// TIA Portal V17 export
// export: Created 2025-03-18T12:31:00.4756631Z, ExportSetting WithDefaults, DisplayName Totally Integrated Automation Portal, DisplayVersion V17 Update 8, DisplayName TIA Portal Openness, DisplayVersion V17 Update 8, DisplayName TIA Portal Version Control Interface, DisplayVersion V17, DisplayName SINAMICS Startdrive Advanced, DisplayVersion V17 SP2, DisplayName SINAMICS Startdrive G110M, G120, G120C, G120D, G120P, G115D, DisplayVersion V17 SP2, DisplayName SINAMICS Startdrive G130, G150, S120, S150, SINAMICS MV, S210, DisplayVersion V17 SP2, DisplayName STEP 7 Professional, DisplayVersion V17 Update 8, DisplayName SINUMERIK ONE STEP 7 Toolbox, DisplayVersion V17 Update 12, DisplayName SINUMERIK 840D sl STEP 7 Toolbox, DisplayVersion V17 Update 12, DisplayName STEP 7 Safety, DisplayVersion V17 Update 6, DisplayName WinCC Advanced, DisplayVersion V17 Update 8
FUNCTION "FC7003_UNIT_01_STATION_04_SAFETY_DOOR" : Void   // FC7003, LAD
{ S7_Optimized_Access := 'FALSE' }
AUTHOR : ETXETAR
VERSION : 1.0
// stored: AutoNumber false, IsIECCheckEnabled false, SetENOAutomatically false, UDAEnableTagReadback false
   VAR_INPUT
      OPTIONS_0 : Byte;   // OPTIONS 0
      CLOSED : Bool;   // CLOSED INPUT
      LOCKED : Bool;   // LOCKED INPUT
   END_VAR
   VAR_OUTPUT
      UNLOCK : Bool;   // UNLOCK OUTPUT
      RED_LIGTH : Bool;   // RED LIGTH OUTPUT
      GREEN_LIGTH : Bool;   // GREEN LIGTH OUTPUT
   END_VAR
   VAR_TEMP
      INPUTS_MASK : Byte;   // INPUTS MASK
      O_BYTE_0 : Struct   // OPTIONS BYTE 0
         IMMEDIATE_STOP : Bool;   // IMMEDIATE STOP REACTION OPTION
         SEOC_WARNING : Bool;   // SEOC WARNING REACTION OPTION
         CLOSED_SENSOR_I : Bool;   // CLOSED SENSOR INPUT OPTION
         CIRCUIT_E2 : Bool;   // CIRCUIT E2 OPTION
         PNEUMATIC_DRIVE : Bool;   // PNEUMATIC DRIVE OPTION
         CHIP_CONVEYOR : Bool;   // CHIP CONVEYOR OPTION
         SPARE_6 : Bool;   // SPARE OPTION
         SPARE_7 : Bool;   // SPARE OPTION
      END_STRUCT;
   END_VAR
   VAR CONSTANT
      FC_NUMBER : DInt := 7003;
   END_VAR
   VAR_TEMP   // added for the SCL form of the ladder/FBD networks
      _w1 : Bool;
      _w2 : Bool;
   END_VAR
BEGIN

REGION Network 1: OPTIONS
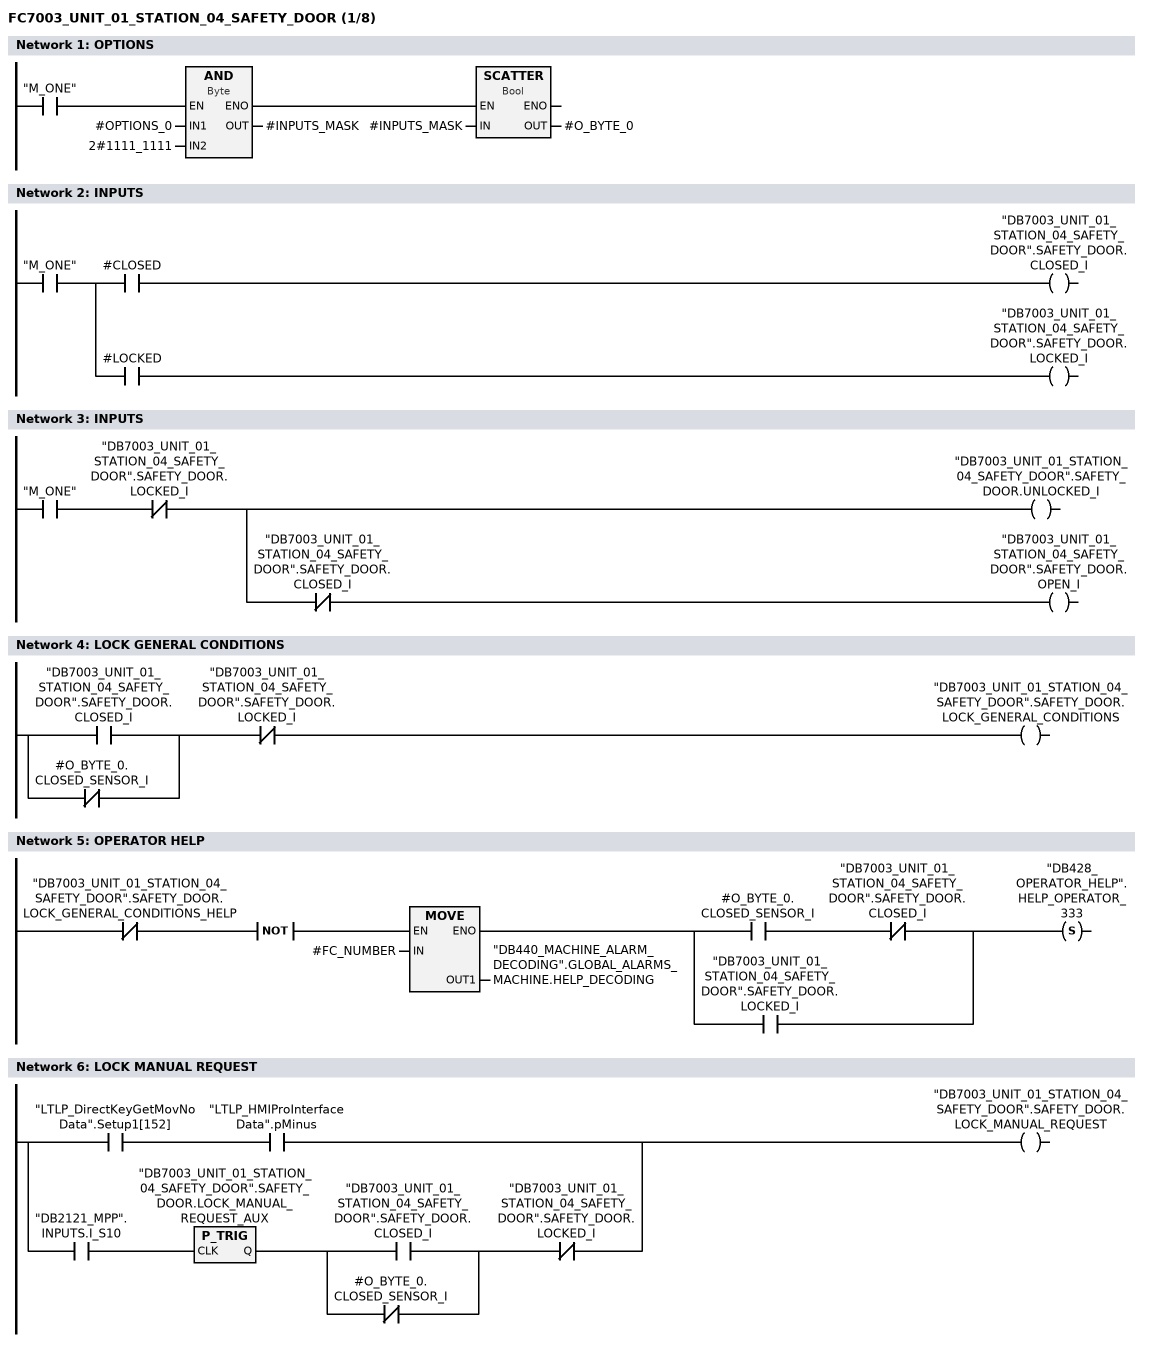
   RUNG wire#powerrail
      Contact( "M_ONE" )
      { S7_Templates := "SrcType := Byte"; S7_GenerateENO := "TRUE" } And(in1 := #OPTIONS_0, in2 := 2#1111_1111, out => #INPUTS_MASK)
      { S7_Templates := "[dest_type := Bool, src_type := Byte]" } SCATTER(IN := #INPUTS_MASK, OUT => #O_BYTE_0)
   END_RUNG
   // the same network as SCL:
   IF "M_ONE" THEN
       #INPUTS_MASK := #OPTIONS_0 AND 2#1111_1111;
       SCATTER(IN := #INPUTS_MASK, OUT => #O_BYTE_0);
   END_IF;
END_REGION

REGION Network 2: INPUTS
   RUNG wire#powerrail
      Contact( "M_ONE" )
      wire#w1
      Contact( #CLOSED )
      Coil( "DB7003_UNIT_01_STATION_04_SAFETY_DOOR".SAFETY_DOOR.CLOSED_I )
   END_RUNG
   RUNG wire#w1
      Contact( #LOCKED )
      Coil( "DB7003_UNIT_01_STATION_04_SAFETY_DOOR".SAFETY_DOOR.LOCKED_I )
   END_RUNG
   // the same network as SCL:
   "DB7003_UNIT_01_STATION_04_SAFETY_DOOR".SAFETY_DOOR.CLOSED_I := "M_ONE" AND #CLOSED;
   "DB7003_UNIT_01_STATION_04_SAFETY_DOOR".SAFETY_DOOR.LOCKED_I := "M_ONE" AND #LOCKED;
END_REGION

REGION Network 3: INPUTS
   RUNG wire#powerrail
      Contact( "M_ONE" )
      I_Contact( "DB7003_UNIT_01_STATION_04_SAFETY_DOOR".SAFETY_DOOR.LOCKED_I )
      wire#w1
      Coil( "DB7003_UNIT_01_STATION_04_SAFETY_DOOR".SAFETY_DOOR.UNLOCKED_I )
   END_RUNG
   RUNG wire#w1
      I_Contact( "DB7003_UNIT_01_STATION_04_SAFETY_DOOR".SAFETY_DOOR.CLOSED_I )
      Coil( "DB7003_UNIT_01_STATION_04_SAFETY_DOOR".SAFETY_DOOR.OPEN_I )
   END_RUNG
   // the same network as SCL:
   "DB7003_UNIT_01_STATION_04_SAFETY_DOOR".SAFETY_DOOR.UNLOCKED_I := "M_ONE" AND NOT "DB7003_UNIT_01_STATION_04_SAFETY_DOOR".SAFETY_DOOR.LOCKED_I;
   "DB7003_UNIT_01_STATION_04_SAFETY_DOOR".SAFETY_DOOR.OPEN_I := "DB7003_UNIT_01_STATION_04_SAFETY_DOOR".SAFETY_DOOR.UNLOCKED_I AND NOT "DB7003_UNIT_01_STATION_04_SAFETY_DOOR".SAFETY_DOOR.CLOSED_I;
END_REGION

REGION Network 4: LOCK GENERAL CONDITIONS
   RUNG wire#powerrail
      Contact( "DB7003_UNIT_01_STATION_04_SAFETY_DOOR".SAFETY_DOOR.CLOSED_I )
      wire#w1
      I_Contact( "DB7003_UNIT_01_STATION_04_SAFETY_DOOR".SAFETY_DOOR.LOCKED_I )
      Coil( "DB7003_UNIT_01_STATION_04_SAFETY_DOOR".SAFETY_DOOR.LOCK_GENERAL_CONDITIONS )
   END_RUNG
   RUNG wire#powerrail
      I_Contact( #O_BYTE_0.CLOSED_SENSOR_I )
   END_RUNG wire#w1
   // the same network as SCL:
   "DB7003_UNIT_01_STATION_04_SAFETY_DOOR".SAFETY_DOOR.LOCK_GENERAL_CONDITIONS := ("DB7003_UNIT_01_STATION_04_SAFETY_DOOR".SAFETY_DOOR.CLOSED_I OR NOT #O_BYTE_0.CLOSED_SENSOR_I) AND NOT "DB7003_UNIT_01_STATION_04_SAFETY_DOOR".SAFETY_DOOR.LOCKED_I;
END_REGION

REGION Network 5: OPERATOR HELP
   RUNG wire#powerrail
      I_Contact( "DB7003_UNIT_01_STATION_04_SAFETY_DOOR".SAFETY_DOOR.LOCK_GENERAL_CONDITIONS_HELP )
      Not()
      { S7_GenerateENO := "TRUE" } Move(in := #FC_NUMBER, out1 => "DB440_MACHINE_ALARM_DECODING".GLOBAL_ALARMS_MACHINE.HELP_DECODING)
      wire#w1
      Contact( #O_BYTE_0.CLOSED_SENSOR_I )
      I_Contact( "DB7003_UNIT_01_STATION_04_SAFETY_DOOR".SAFETY_DOOR.CLOSED_I )
      wire#w2
      S_Coil( "DB428_OPERATOR_HELP".HELP_OPERATOR_333 )
   END_RUNG
   RUNG wire#w1
      Contact( "DB7003_UNIT_01_STATION_04_SAFETY_DOOR".SAFETY_DOOR.LOCKED_I )
   END_RUNG wire#w2
   // the same network as SCL:
   // ENO of a box is taken as its EN; it also drops when the box reports an error
   #_w1 := NOT (NOT "DB7003_UNIT_01_STATION_04_SAFETY_DOOR".SAFETY_DOOR.LOCK_GENERAL_CONDITIONS_HELP);
   IF #_w1 THEN "DB440_MACHINE_ALARM_DECODING".GLOBAL_ALARMS_MACHINE.HELP_DECODING := #FC_NUMBER; END_IF;
   IF #_w1 AND ((#O_BYTE_0.CLOSED_SENSOR_I AND NOT "DB7003_UNIT_01_STATION_04_SAFETY_DOOR".SAFETY_DOOR.CLOSED_I) OR "DB7003_UNIT_01_STATION_04_SAFETY_DOOR".SAFETY_DOOR.LOCKED_I) THEN
       "DB428_OPERATOR_HELP".HELP_OPERATOR_333 := TRUE;
   END_IF;
END_REGION

REGION Network 6: LOCK MANUAL REQUEST
   RUNG wire#powerrail
      Contact( "LTLP_DirectKeyGetMovNoData".Setup1[152] )
      Contact( "LTLP_HMIProInterfaceData".pMinus )
      wire#w1
      Coil( "DB7003_UNIT_01_STATION_04_SAFETY_DOOR".SAFETY_DOOR.LOCK_MANUAL_REQUEST )
   END_RUNG
   RUNG wire#powerrail
      Contact( "DB2121_MPP".INPUTS.I_S10 )
      P_Trig( "DB7003_UNIT_01_STATION_04_SAFETY_DOOR".SAFETY_DOOR.LOCK_MANUAL_REQUEST_AUX )
      wire#w2
      Contact( "DB7003_UNIT_01_STATION_04_SAFETY_DOOR".SAFETY_DOOR.CLOSED_I )
      wire#w3
      I_Contact( "DB7003_UNIT_01_STATION_04_SAFETY_DOOR".SAFETY_DOOR.LOCKED_I )
   END_RUNG wire#w1
   RUNG wire#w2
      I_Contact( #O_BYTE_0.CLOSED_SENSOR_I )
   END_RUNG wire#w3
   // the same network as SCL:
   #_w1 := "DB2121_MPP".INPUTS.I_S10 AND NOT "DB7003_UNIT_01_STATION_04_SAFETY_DOOR".SAFETY_DOOR.LOCK_MANUAL_REQUEST_AUX;   // rising edge
   "DB7003_UNIT_01_STATION_04_SAFETY_DOOR".SAFETY_DOOR.LOCK_MANUAL_REQUEST_AUX := "DB2121_MPP".INPUTS.I_S10;
   "DB7003_UNIT_01_STATION_04_SAFETY_DOOR".SAFETY_DOOR.LOCK_MANUAL_REQUEST := ("LTLP_DirectKeyGetMovNoData".Setup1[152] AND "LTLP_HMIProInterfaceData".pMinus) OR (#_w1 AND ("DB7003_UNIT_01_STATION_04_SAFETY_DOOR".SAFETY_DOOR.CLOSED_I OR NOT #O_BYTE_0.CLOSED_SENSOR_I) AND NOT "DB7003_UNIT_01_STATION_04_SAFETY_DOOR".SAFETY_DOOR.LOCKED_I);
END_REGION

REGION Network 7: LOCK AUTO REQUEST
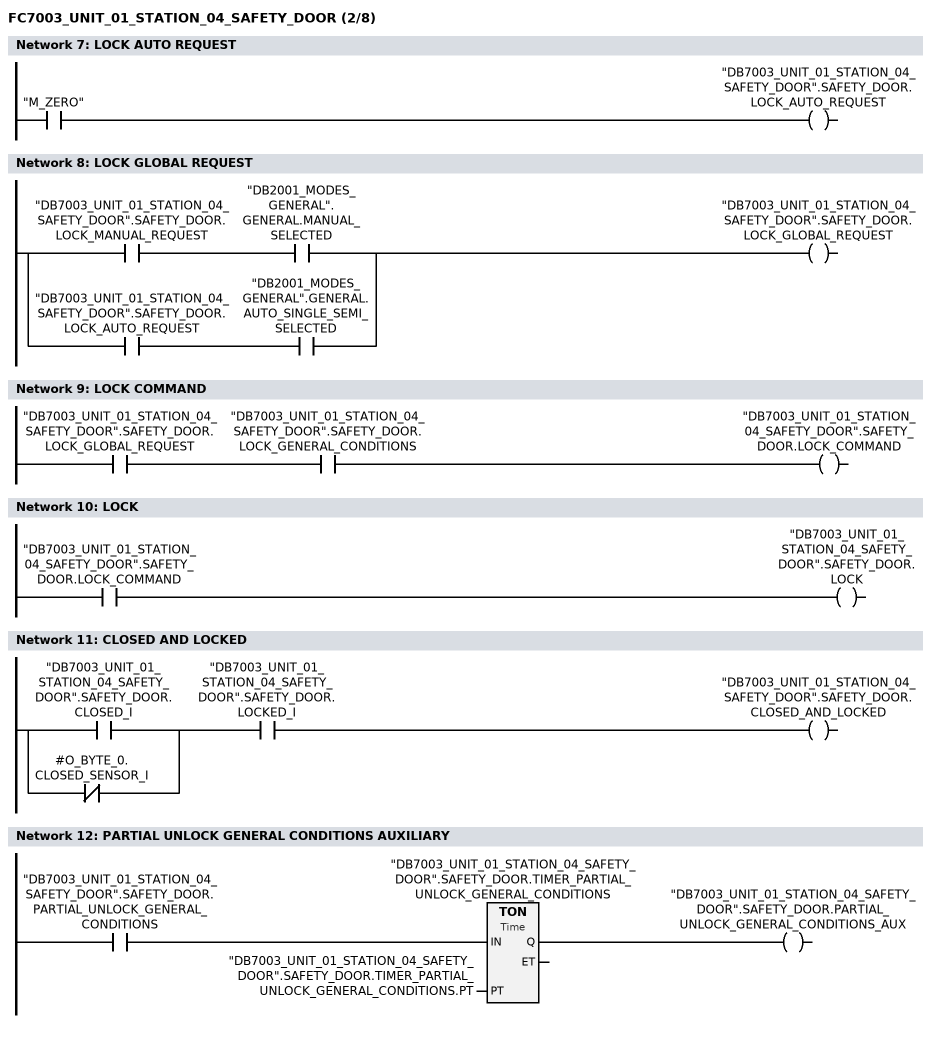
   RUNG wire#powerrail
      Contact( "M_ZERO" )
      Coil( "DB7003_UNIT_01_STATION_04_SAFETY_DOOR".SAFETY_DOOR.LOCK_AUTO_REQUEST )
   END_RUNG
   // the same network as SCL:
   "DB7003_UNIT_01_STATION_04_SAFETY_DOOR".SAFETY_DOOR.LOCK_AUTO_REQUEST := "M_ZERO";
END_REGION

REGION Network 8: LOCK GLOBAL REQUEST
   RUNG wire#powerrail
      Contact( "DB7003_UNIT_01_STATION_04_SAFETY_DOOR".SAFETY_DOOR.LOCK_MANUAL_REQUEST )
      Contact( "DB2001_MODES_GENERAL".GENERAL.MANUAL_SELECTED )
      wire#w1
      Coil( "DB7003_UNIT_01_STATION_04_SAFETY_DOOR".SAFETY_DOOR.LOCK_GLOBAL_REQUEST )
   END_RUNG
   RUNG wire#powerrail
      Contact( "DB7003_UNIT_01_STATION_04_SAFETY_DOOR".SAFETY_DOOR.LOCK_AUTO_REQUEST )
      Contact( "DB2001_MODES_GENERAL".GENERAL.AUTO_SINGLE_SEMI_SELECTED )
   END_RUNG wire#w1
   // the same network as SCL:
   "DB7003_UNIT_01_STATION_04_SAFETY_DOOR".SAFETY_DOOR.LOCK_GLOBAL_REQUEST := ("DB7003_UNIT_01_STATION_04_SAFETY_DOOR".SAFETY_DOOR.LOCK_MANUAL_REQUEST AND "DB2001_MODES_GENERAL".GENERAL.MANUAL_SELECTED) OR ("DB7003_UNIT_01_STATION_04_SAFETY_DOOR".SAFETY_DOOR.LOCK_AUTO_REQUEST AND "DB2001_MODES_GENERAL".GENERAL.AUTO_SINGLE_SEMI_SELECTED);
END_REGION

REGION Network 9: LOCK COMMAND
   RUNG wire#powerrail
      Contact( "DB7003_UNIT_01_STATION_04_SAFETY_DOOR".SAFETY_DOOR.LOCK_GLOBAL_REQUEST )
      Contact( "DB7003_UNIT_01_STATION_04_SAFETY_DOOR".SAFETY_DOOR.LOCK_GENERAL_CONDITIONS )
      Coil( "DB7003_UNIT_01_STATION_04_SAFETY_DOOR".SAFETY_DOOR.LOCK_COMMAND )
   END_RUNG
   // the same network as SCL:
   "DB7003_UNIT_01_STATION_04_SAFETY_DOOR".SAFETY_DOOR.LOCK_COMMAND := "DB7003_UNIT_01_STATION_04_SAFETY_DOOR".SAFETY_DOOR.LOCK_GLOBAL_REQUEST AND "DB7003_UNIT_01_STATION_04_SAFETY_DOOR".SAFETY_DOOR.LOCK_GENERAL_CONDITIONS;
END_REGION

REGION Network 10: LOCK
   RUNG wire#powerrail
      Contact( "DB7003_UNIT_01_STATION_04_SAFETY_DOOR".SAFETY_DOOR.LOCK_COMMAND )
      Coil( "DB7003_UNIT_01_STATION_04_SAFETY_DOOR".SAFETY_DOOR.LOCK )
   END_RUNG
   // the same network as SCL:
   "DB7003_UNIT_01_STATION_04_SAFETY_DOOR".SAFETY_DOOR.LOCK := "DB7003_UNIT_01_STATION_04_SAFETY_DOOR".SAFETY_DOOR.LOCK_COMMAND;
END_REGION

REGION Network 11: CLOSED AND LOCKED
   RUNG wire#powerrail
      Contact( "DB7003_UNIT_01_STATION_04_SAFETY_DOOR".SAFETY_DOOR.CLOSED_I )
      wire#w1
      Contact( "DB7003_UNIT_01_STATION_04_SAFETY_DOOR".SAFETY_DOOR.LOCKED_I )
      Coil( "DB7003_UNIT_01_STATION_04_SAFETY_DOOR".SAFETY_DOOR.CLOSED_AND_LOCKED )
   END_RUNG
   RUNG wire#powerrail
      I_Contact( #O_BYTE_0.CLOSED_SENSOR_I )
   END_RUNG wire#w1
   // the same network as SCL:
   "DB7003_UNIT_01_STATION_04_SAFETY_DOOR".SAFETY_DOOR.CLOSED_AND_LOCKED := ("DB7003_UNIT_01_STATION_04_SAFETY_DOOR".SAFETY_DOOR.CLOSED_I OR NOT #O_BYTE_0.CLOSED_SENSOR_I) AND "DB7003_UNIT_01_STATION_04_SAFETY_DOOR".SAFETY_DOOR.LOCKED_I;
END_REGION

REGION Network 12: PARTIAL UNLOCK GENERAL CONDITIONS AUXILIARY
   RUNG wire#powerrail
      Contact( "DB7003_UNIT_01_STATION_04_SAFETY_DOOR".SAFETY_DOOR.PARTIAL_UNLOCK_GENERAL_CONDITIONS )
      { S7_Templates := "time_type := Time" } "DB7003_UNIT_01_STATION_04_SAFETY_DOOR".SAFETY_DOOR.TIMER_PARTIAL_UNLOCK_GENERAL_CONDITIONS.TON(pt := "DB7003_UNIT_01_STATION_04_SAFETY_DOOR".SAFETY_DOOR.TIMER_PARTIAL_UNLOCK_GENERAL_CONDITIONS.PT, et =>)
      Coil( "DB7003_UNIT_01_STATION_04_SAFETY_DOOR".SAFETY_DOOR.PARTIAL_UNLOCK_GENERAL_CONDITIONS_AUX )
   END_RUNG
   // the same network as SCL:
   "DB7003_UNIT_01_STATION_04_SAFETY_DOOR".SAFETY_DOOR.TIMER_PARTIAL_UNLOCK_GENERAL_CONDITIONS.TON(IN := "DB7003_UNIT_01_STATION_04_SAFETY_DOOR".SAFETY_DOOR.PARTIAL_UNLOCK_GENERAL_CONDITIONS,
                           PT := "DB7003_UNIT_01_STATION_04_SAFETY_DOOR".SAFETY_DOOR.TIMER_PARTIAL_UNLOCK_GENERAL_CONDITIONS.PT);
   "DB7003_UNIT_01_STATION_04_SAFETY_DOOR".SAFETY_DOOR.PARTIAL_UNLOCK_GENERAL_CONDITIONS_AUX := "DB7003_UNIT_01_STATION_04_SAFETY_DOOR".SAFETY_DOOR.TIMER_PARTIAL_UNLOCK_GENERAL_CONDITIONS.Q;
END_REGION

REGION Network 13: UNLOCK GENERAL CONDITIONS
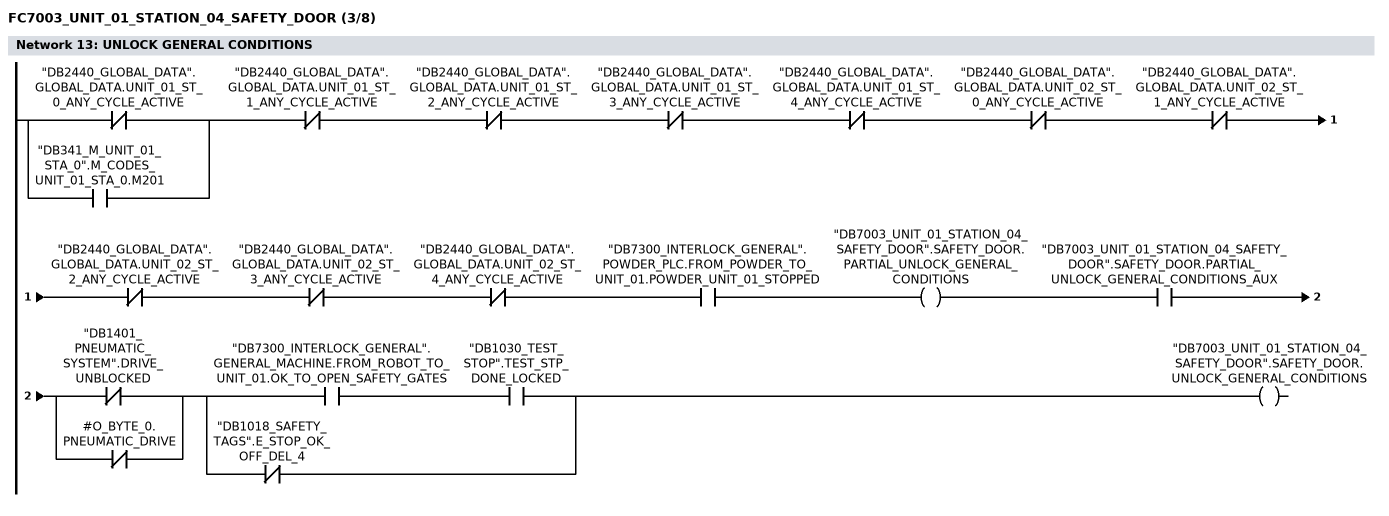
   RUNG wire#powerrail
      I_Contact( "DB2440_GLOBAL_DATA".GLOBAL_DATA.UNIT_01_ST_0_ANY_CYCLE_ACTIVE )
      wire#w1
      I_Contact( "DB2440_GLOBAL_DATA".GLOBAL_DATA.UNIT_01_ST_1_ANY_CYCLE_ACTIVE )
      I_Contact( "DB2440_GLOBAL_DATA".GLOBAL_DATA.UNIT_01_ST_2_ANY_CYCLE_ACTIVE )
      I_Contact( "DB2440_GLOBAL_DATA".GLOBAL_DATA.UNIT_01_ST_3_ANY_CYCLE_ACTIVE )
      I_Contact( "DB2440_GLOBAL_DATA".GLOBAL_DATA.UNIT_01_ST_4_ANY_CYCLE_ACTIVE )
      I_Contact( "DB2440_GLOBAL_DATA".GLOBAL_DATA.UNIT_02_ST_0_ANY_CYCLE_ACTIVE )
      I_Contact( "DB2440_GLOBAL_DATA".GLOBAL_DATA.UNIT_02_ST_1_ANY_CYCLE_ACTIVE )
      I_Contact( "DB2440_GLOBAL_DATA".GLOBAL_DATA.UNIT_02_ST_2_ANY_CYCLE_ACTIVE )
      I_Contact( "DB2440_GLOBAL_DATA".GLOBAL_DATA.UNIT_02_ST_3_ANY_CYCLE_ACTIVE )
      I_Contact( "DB2440_GLOBAL_DATA".GLOBAL_DATA.UNIT_02_ST_4_ANY_CYCLE_ACTIVE )
      Contact( "DB7300_INTERLOCK_GENERAL".POWDER_PLC.FROM_POWDER_TO_UNIT_01.POWDER_UNIT_01_STOPPED )
      Coil( "DB7003_UNIT_01_STATION_04_SAFETY_DOOR".SAFETY_DOOR.PARTIAL_UNLOCK_GENERAL_CONDITIONS )
      Contact( "DB7003_UNIT_01_STATION_04_SAFETY_DOOR".SAFETY_DOOR.PARTIAL_UNLOCK_GENERAL_CONDITIONS_AUX )
      wire#w2
      I_Contact( "DB1401_PNEUMATIC_SYSTEM".DRIVE_UNBLOCKED )
      wire#w3
      Contact( "DB7300_INTERLOCK_GENERAL".GENERAL_MACHINE.FROM_ROBOT_TO_UNIT_01.OK_TO_OPEN_SAFETY_GATES )
      Contact( "DB1030_TEST_STOP".TEST_STP_DONE_LOCKED )
      wire#w4
      Coil( "DB7003_UNIT_01_STATION_04_SAFETY_DOOR".SAFETY_DOOR.UNLOCK_GENERAL_CONDITIONS )
   END_RUNG
   RUNG wire#powerrail
      Contact( "DB341_M_UNIT_01_STA_0".M_CODES_UNIT_01_STA_0.M201 )
   END_RUNG wire#w1
   RUNG wire#w2
      I_Contact( #O_BYTE_0.PNEUMATIC_DRIVE )
   END_RUNG wire#w3
   RUNG wire#w3
      I_Contact( "DB1018_SAFETY_TAGS".E_STOP_OK_OFF_DEL_4 )
   END_RUNG wire#w4
   // the same network as SCL:
   "DB7003_UNIT_01_STATION_04_SAFETY_DOOR".SAFETY_DOOR.PARTIAL_UNLOCK_GENERAL_CONDITIONS := (NOT "DB2440_GLOBAL_DATA".GLOBAL_DATA.UNIT_01_ST_0_ANY_CYCLE_ACTIVE OR "DB341_M_UNIT_01_STA_0".M_CODES_UNIT_01_STA_0.M201) AND NOT "DB2440_GLOBAL_DATA".GLOBAL_DATA.UNIT_01_ST_1_ANY_CYCLE_ACTIVE AND NOT "DB2440_GLOBAL_DATA".GLOBAL_DATA.UNIT_01_ST_2_ANY_CYCLE_ACTIVE AND NOT "DB2440_GLOBAL_DATA".GLOBAL_DATA.UNIT_01_ST_3_ANY_CYCLE_ACTIVE AND NOT "DB2440_GLOBAL_DATA".GLOBAL_DATA.UNIT_01_ST_4_ANY_CYCLE_ACTIVE AND NOT "DB2440_GLOBAL_DATA".GLOBAL_DATA.UNIT_02_ST_0_ANY_CYCLE_ACTIVE AND NOT "DB2440_GLOBAL_DATA".GLOBAL_DATA.UNIT_02_ST_1_ANY_CYCLE_ACTIVE AND NOT "DB2440_GLOBAL_DATA".GLOBAL_DATA.UNIT_02_ST_2_ANY_CYCLE_ACTIVE AND NOT "DB2440_GLOBAL_DATA".GLOBAL_DATA.UNIT_02_ST_3_ANY_CYCLE_ACTIVE AND NOT "DB2440_GLOBAL_DATA".GLOBAL_DATA.UNIT_02_ST_4_ANY_CYCLE_ACTIVE AND "DB7300_INTERLOCK_GENERAL".POWDER_PLC.FROM_POWDER_TO_UNIT_01.POWDER_UNIT_01_STOPPED;
   "DB7003_UNIT_01_STATION_04_SAFETY_DOOR".SAFETY_DOOR.UNLOCK_GENERAL_CONDITIONS := "DB7003_UNIT_01_STATION_04_SAFETY_DOOR".SAFETY_DOOR.PARTIAL_UNLOCK_GENERAL_CONDITIONS AND "DB7003_UNIT_01_STATION_04_SAFETY_DOOR".SAFETY_DOOR.PARTIAL_UNLOCK_GENERAL_CONDITIONS_AUX AND (NOT "DB1401_PNEUMATIC_SYSTEM".DRIVE_UNBLOCKED OR NOT #O_BYTE_0.PNEUMATIC_DRIVE) AND (("DB7300_INTERLOCK_GENERAL".GENERAL_MACHINE.FROM_ROBOT_TO_UNIT_01.OK_TO_OPEN_SAFETY_GATES AND "DB1030_TEST_STOP".TEST_STP_DONE_LOCKED) OR NOT "DB1018_SAFETY_TAGS".E_STOP_OK_OFF_DEL_4);
END_REGION

REGION Network 14: OPERATOR HELP
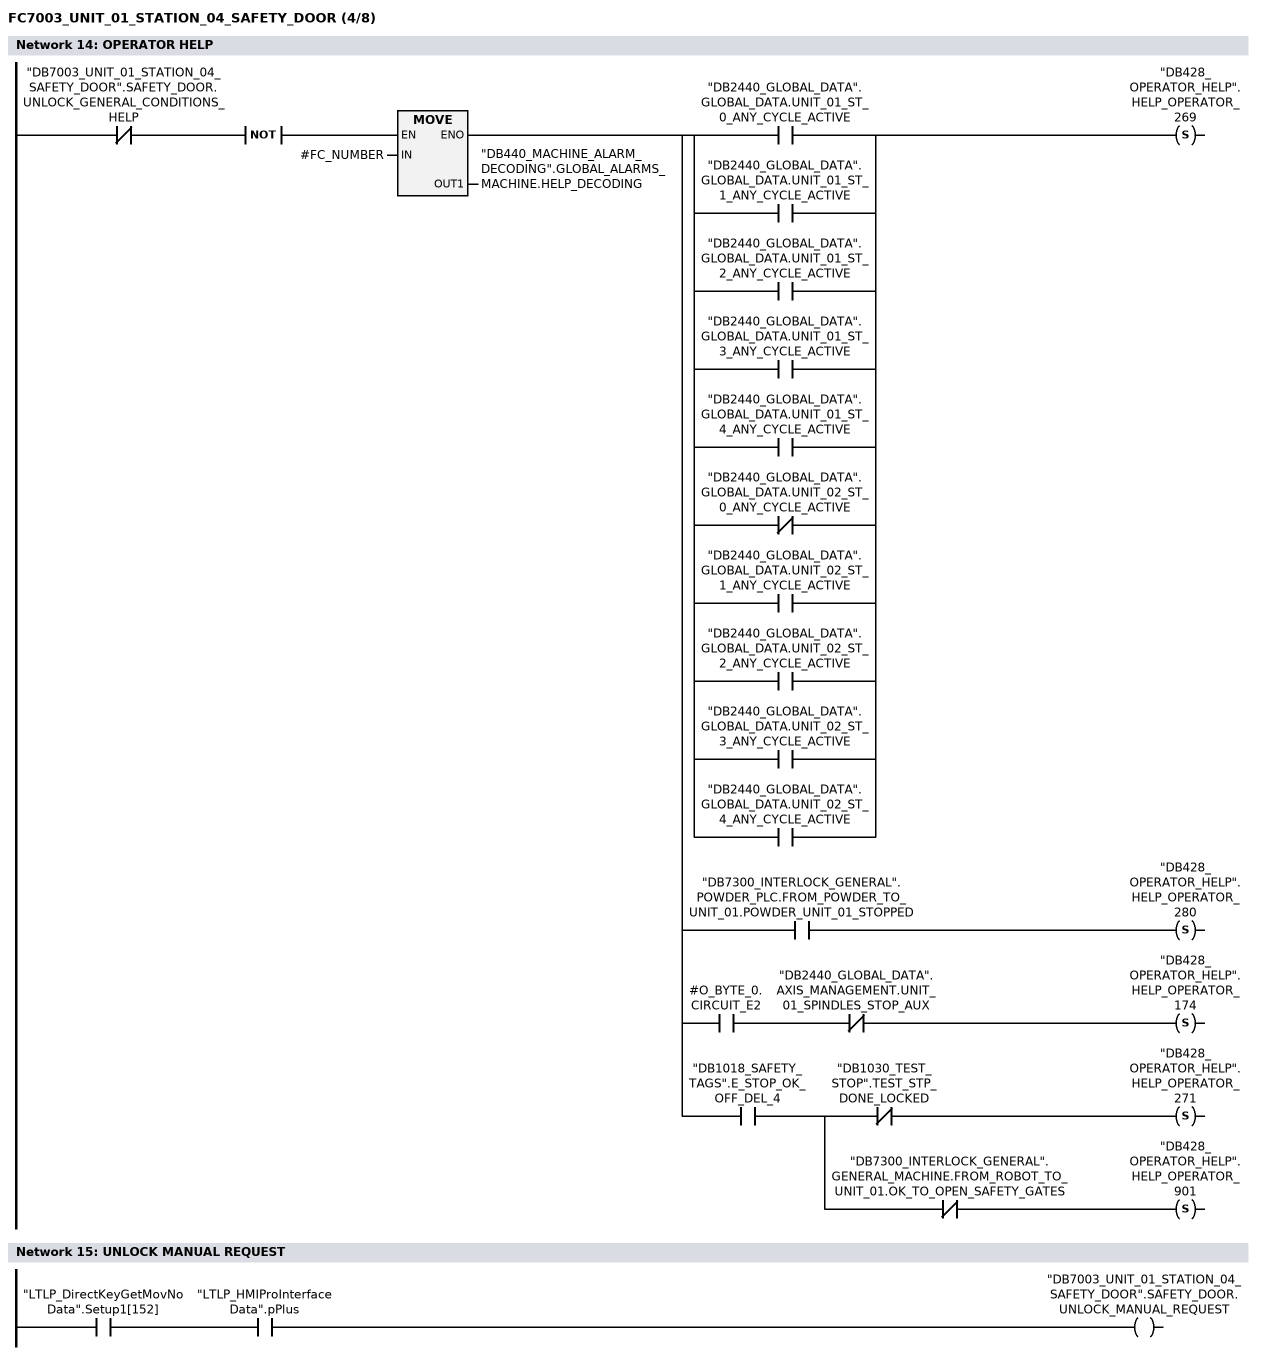
   RUNG wire#powerrail
      I_Contact( "DB7003_UNIT_01_STATION_04_SAFETY_DOOR".SAFETY_DOOR.UNLOCK_GENERAL_CONDITIONS_HELP )
      Not()
      { S7_GenerateENO := "TRUE" } Move(in := #FC_NUMBER, out1 => "DB440_MACHINE_ALARM_DECODING".GLOBAL_ALARMS_MACHINE.HELP_DECODING)
      wire#w1
      Contact( "DB2440_GLOBAL_DATA".GLOBAL_DATA.UNIT_01_ST_0_ANY_CYCLE_ACTIVE )
      wire#w2
      S_Coil( "DB428_OPERATOR_HELP".HELP_OPERATOR_269 )
   END_RUNG
   RUNG wire#w1
      Contact( "DB2440_GLOBAL_DATA".GLOBAL_DATA.UNIT_01_ST_1_ANY_CYCLE_ACTIVE )
   END_RUNG wire#w2
   RUNG wire#w1
      Contact( "DB2440_GLOBAL_DATA".GLOBAL_DATA.UNIT_01_ST_2_ANY_CYCLE_ACTIVE )
   END_RUNG wire#w2
   RUNG wire#w1
      Contact( "DB2440_GLOBAL_DATA".GLOBAL_DATA.UNIT_01_ST_3_ANY_CYCLE_ACTIVE )
   END_RUNG wire#w2
   RUNG wire#w1
      Contact( "DB2440_GLOBAL_DATA".GLOBAL_DATA.UNIT_01_ST_4_ANY_CYCLE_ACTIVE )
   END_RUNG wire#w2
   RUNG wire#w1
      I_Contact( "DB2440_GLOBAL_DATA".GLOBAL_DATA.UNIT_02_ST_0_ANY_CYCLE_ACTIVE )
   END_RUNG wire#w2
   RUNG wire#w1
      Contact( "DB2440_GLOBAL_DATA".GLOBAL_DATA.UNIT_02_ST_1_ANY_CYCLE_ACTIVE )
   END_RUNG wire#w2
   RUNG wire#w1
      Contact( "DB2440_GLOBAL_DATA".GLOBAL_DATA.UNIT_02_ST_2_ANY_CYCLE_ACTIVE )
   END_RUNG wire#w2
   RUNG wire#w1
      Contact( "DB2440_GLOBAL_DATA".GLOBAL_DATA.UNIT_02_ST_3_ANY_CYCLE_ACTIVE )
   END_RUNG wire#w2
   RUNG wire#w1
      Contact( "DB2440_GLOBAL_DATA".GLOBAL_DATA.UNIT_02_ST_4_ANY_CYCLE_ACTIVE )
   END_RUNG wire#w2
   RUNG wire#w1
      Contact( "DB7300_INTERLOCK_GENERAL".POWDER_PLC.FROM_POWDER_TO_UNIT_01.POWDER_UNIT_01_STOPPED )
      S_Coil( "DB428_OPERATOR_HELP".HELP_OPERATOR_280 )
   END_RUNG
   RUNG wire#w1
      Contact( #O_BYTE_0.CIRCUIT_E2 )
      I_Contact( "DB2440_GLOBAL_DATA".AXIS_MANAGEMENT.UNIT_01_SPINDLES_STOP_AUX )
      S_Coil( "DB428_OPERATOR_HELP".HELP_OPERATOR_174 )
   END_RUNG
   RUNG wire#w1
      Contact( "DB1018_SAFETY_TAGS".E_STOP_OK_OFF_DEL_4 )
      wire#w3
      I_Contact( "DB1030_TEST_STOP".TEST_STP_DONE_LOCKED )
      S_Coil( "DB428_OPERATOR_HELP".HELP_OPERATOR_271 )
   END_RUNG
   RUNG wire#w3
      I_Contact( "DB7300_INTERLOCK_GENERAL".GENERAL_MACHINE.FROM_ROBOT_TO_UNIT_01.OK_TO_OPEN_SAFETY_GATES )
      S_Coil( "DB428_OPERATOR_HELP".HELP_OPERATOR_901 )
   END_RUNG
   // the same network as SCL:
   // ENO of a box is taken as its EN; it also drops when the box reports an error
   #_w1 := NOT (NOT "DB7003_UNIT_01_STATION_04_SAFETY_DOOR".SAFETY_DOOR.UNLOCK_GENERAL_CONDITIONS_HELP);
   IF #_w1 THEN "DB440_MACHINE_ALARM_DECODING".GLOBAL_ALARMS_MACHINE.HELP_DECODING := #FC_NUMBER; END_IF;
   IF #_w1 AND ("DB2440_GLOBAL_DATA".GLOBAL_DATA.UNIT_01_ST_0_ANY_CYCLE_ACTIVE OR "DB2440_GLOBAL_DATA".GLOBAL_DATA.UNIT_01_ST_1_ANY_CYCLE_ACTIVE OR "DB2440_GLOBAL_DATA".GLOBAL_DATA.UNIT_01_ST_2_ANY_CYCLE_ACTIVE OR "DB2440_GLOBAL_DATA".GLOBAL_DATA.UNIT_01_ST_3_ANY_CYCLE_ACTIVE OR "DB2440_GLOBAL_DATA".GLOBAL_DATA.UNIT_01_ST_4_ANY_CYCLE_ACTIVE OR NOT "DB2440_GLOBAL_DATA".GLOBAL_DATA.UNIT_02_ST_0_ANY_CYCLE_ACTIVE OR "DB2440_GLOBAL_DATA".GLOBAL_DATA.UNIT_02_ST_1_ANY_CYCLE_ACTIVE OR "DB2440_GLOBAL_DATA".GLOBAL_DATA.UNIT_02_ST_2_ANY_CYCLE_ACTIVE OR "DB2440_GLOBAL_DATA".GLOBAL_DATA.UNIT_02_ST_3_ANY_CYCLE_ACTIVE OR "DB2440_GLOBAL_DATA".GLOBAL_DATA.UNIT_02_ST_4_ANY_CYCLE_ACTIVE) THEN
       "DB428_OPERATOR_HELP".HELP_OPERATOR_269 := TRUE;
   END_IF;
   IF #_w1 AND "DB7300_INTERLOCK_GENERAL".POWDER_PLC.FROM_POWDER_TO_UNIT_01.POWDER_UNIT_01_STOPPED THEN
       "DB428_OPERATOR_HELP".HELP_OPERATOR_280 := TRUE;
   END_IF;
   IF #_w1 AND #O_BYTE_0.CIRCUIT_E2 AND NOT "DB2440_GLOBAL_DATA".AXIS_MANAGEMENT.UNIT_01_SPINDLES_STOP_AUX THEN
       "DB428_OPERATOR_HELP".HELP_OPERATOR_174 := TRUE;
   END_IF;
   #_w2 := #_w1 AND "DB1018_SAFETY_TAGS".E_STOP_OK_OFF_DEL_4;
   IF #_w2 AND NOT "DB1030_TEST_STOP".TEST_STP_DONE_LOCKED THEN
       "DB428_OPERATOR_HELP".HELP_OPERATOR_271 := TRUE;
   END_IF;
   IF #_w2 AND NOT "DB7300_INTERLOCK_GENERAL".GENERAL_MACHINE.FROM_ROBOT_TO_UNIT_01.OK_TO_OPEN_SAFETY_GATES THEN
       "DB428_OPERATOR_HELP".HELP_OPERATOR_901 := TRUE;
   END_IF;
END_REGION

REGION Network 15: UNLOCK MANUAL REQUEST
   RUNG wire#powerrail
      Contact( "LTLP_DirectKeyGetMovNoData".Setup1[152] )
      Contact( "LTLP_HMIProInterfaceData".pPlus )
      Coil( "DB7003_UNIT_01_STATION_04_SAFETY_DOOR".SAFETY_DOOR.UNLOCK_MANUAL_REQUEST )
   END_RUNG
   // the same network as SCL:
   "DB7003_UNIT_01_STATION_04_SAFETY_DOOR".SAFETY_DOOR.UNLOCK_MANUAL_REQUEST := "LTLP_DirectKeyGetMovNoData".Setup1[152] AND "LTLP_HMIProInterfaceData".pPlus;
END_REGION

REGION Network 16: OPERATOR HELP
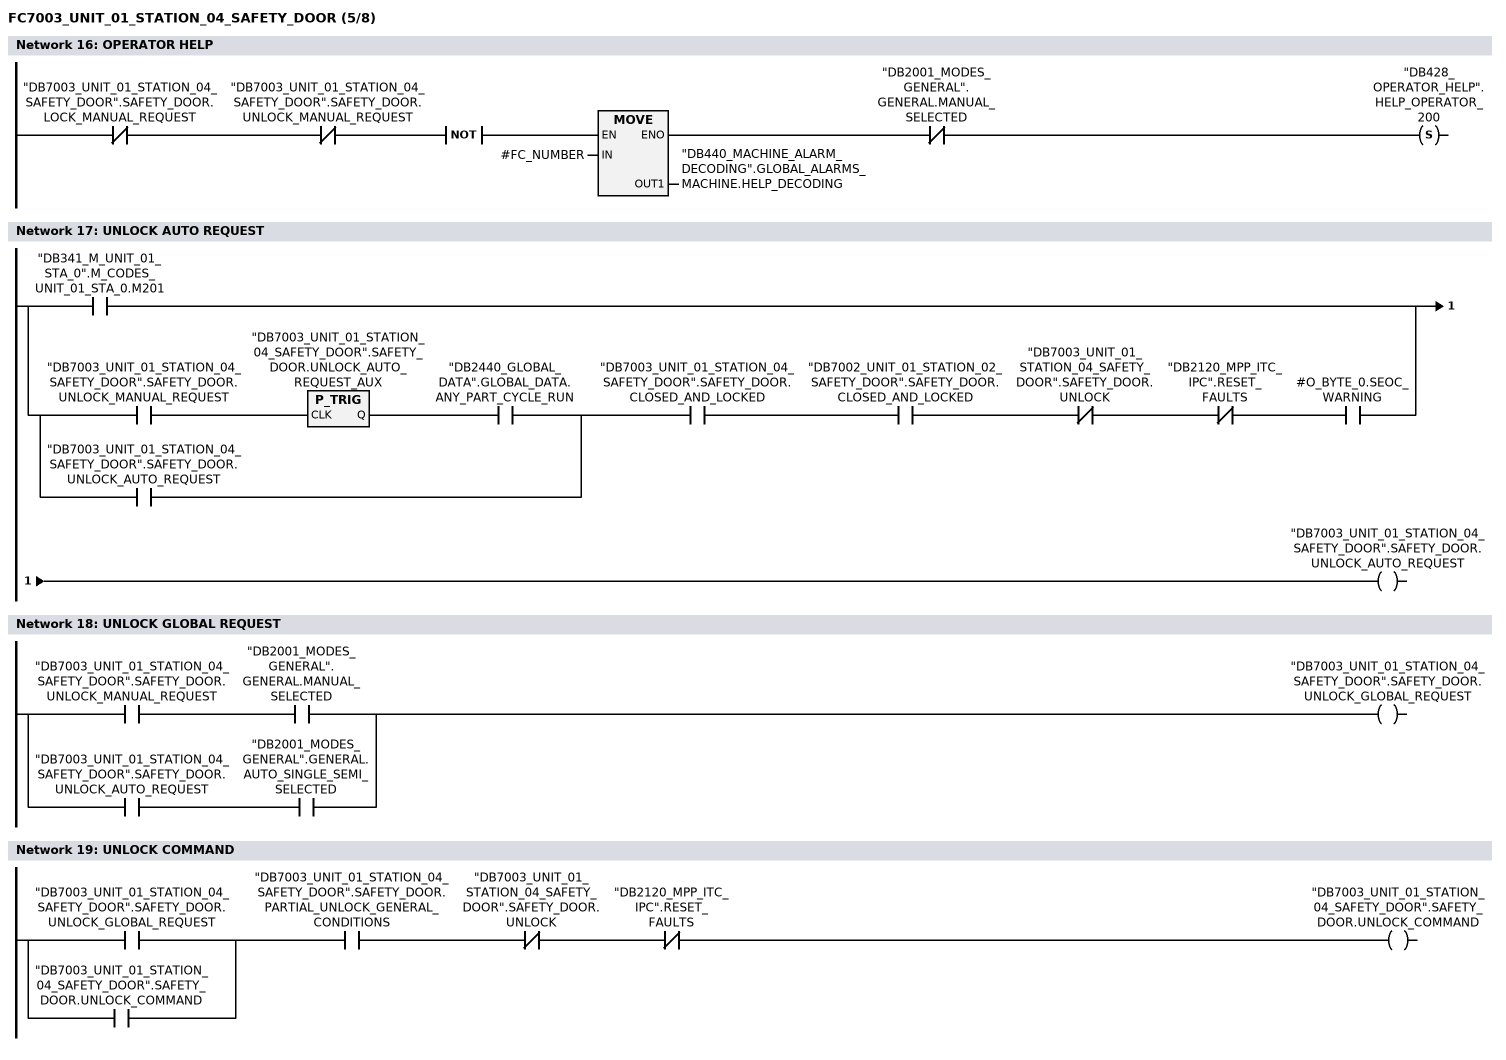
   RUNG wire#powerrail
      I_Contact( "DB7003_UNIT_01_STATION_04_SAFETY_DOOR".SAFETY_DOOR.LOCK_MANUAL_REQUEST )
      I_Contact( "DB7003_UNIT_01_STATION_04_SAFETY_DOOR".SAFETY_DOOR.UNLOCK_MANUAL_REQUEST )
      Not()
      { S7_GenerateENO := "TRUE" } Move(in := #FC_NUMBER, out1 => "DB440_MACHINE_ALARM_DECODING".GLOBAL_ALARMS_MACHINE.HELP_DECODING)
      I_Contact( "DB2001_MODES_GENERAL".GENERAL.MANUAL_SELECTED )
      S_Coil( "DB428_OPERATOR_HELP".HELP_OPERATOR_200 )
   END_RUNG
   // the same network as SCL:
   // ENO of a box is taken as its EN; it also drops when the box reports an error
   #_w1 := NOT (NOT "DB7003_UNIT_01_STATION_04_SAFETY_DOOR".SAFETY_DOOR.LOCK_MANUAL_REQUEST AND NOT "DB7003_UNIT_01_STATION_04_SAFETY_DOOR".SAFETY_DOOR.UNLOCK_MANUAL_REQUEST);
   IF #_w1 THEN "DB440_MACHINE_ALARM_DECODING".GLOBAL_ALARMS_MACHINE.HELP_DECODING := #FC_NUMBER; END_IF;
   IF #_w1 AND NOT "DB2001_MODES_GENERAL".GENERAL.MANUAL_SELECTED THEN
       "DB428_OPERATOR_HELP".HELP_OPERATOR_200 := TRUE;
   END_IF;
END_REGION

REGION Network 17: UNLOCK AUTO REQUEST
   RUNG wire#powerrail
      Contact( "DB341_M_UNIT_01_STA_0".M_CODES_UNIT_01_STA_0.M201 )
      wire#w1
      Coil( "DB7003_UNIT_01_STATION_04_SAFETY_DOOR".SAFETY_DOOR.UNLOCK_AUTO_REQUEST )
   END_RUNG
   RUNG wire#powerrail
      Contact( "DB7003_UNIT_01_STATION_04_SAFETY_DOOR".SAFETY_DOOR.UNLOCK_MANUAL_REQUEST )
      P_Trig( "DB7003_UNIT_01_STATION_04_SAFETY_DOOR".SAFETY_DOOR.UNLOCK_AUTO_REQUEST_AUX )
      Contact( "DB2440_GLOBAL_DATA".GLOBAL_DATA.ANY_PART_CYCLE_RUN )
      wire#w2
      Contact( "DB7003_UNIT_01_STATION_04_SAFETY_DOOR".SAFETY_DOOR.CLOSED_AND_LOCKED )
      Contact( "DB7002_UNIT_01_STATION_02_SAFETY_DOOR".SAFETY_DOOR.CLOSED_AND_LOCKED )
      I_Contact( "DB7003_UNIT_01_STATION_04_SAFETY_DOOR".SAFETY_DOOR.UNLOCK )
      I_Contact( "DB2120_MPP_ITC_IPC".RESET_FAULTS )
      Contact( #O_BYTE_0.SEOC_WARNING )
   END_RUNG wire#w1
   RUNG wire#powerrail
      Contact( "DB7003_UNIT_01_STATION_04_SAFETY_DOOR".SAFETY_DOOR.UNLOCK_AUTO_REQUEST )
   END_RUNG wire#w2
   // the same network as SCL:
   #_w1 := "DB7003_UNIT_01_STATION_04_SAFETY_DOOR".SAFETY_DOOR.UNLOCK_MANUAL_REQUEST AND NOT "DB7003_UNIT_01_STATION_04_SAFETY_DOOR".SAFETY_DOOR.UNLOCK_AUTO_REQUEST_AUX;   // rising edge
   "DB7003_UNIT_01_STATION_04_SAFETY_DOOR".SAFETY_DOOR.UNLOCK_AUTO_REQUEST_AUX := "DB7003_UNIT_01_STATION_04_SAFETY_DOOR".SAFETY_DOOR.UNLOCK_MANUAL_REQUEST;
   "DB7003_UNIT_01_STATION_04_SAFETY_DOOR".SAFETY_DOOR.UNLOCK_AUTO_REQUEST := "DB341_M_UNIT_01_STA_0".M_CODES_UNIT_01_STA_0.M201 OR (((#_w1 AND "DB2440_GLOBAL_DATA".GLOBAL_DATA.ANY_PART_CYCLE_RUN) OR "DB7003_UNIT_01_STATION_04_SAFETY_DOOR".SAFETY_DOOR.UNLOCK_AUTO_REQUEST) AND "DB7003_UNIT_01_STATION_04_SAFETY_DOOR".SAFETY_DOOR.CLOSED_AND_LOCKED AND "DB7002_UNIT_01_STATION_02_SAFETY_DOOR".SAFETY_DOOR.CLOSED_AND_LOCKED AND NOT "DB7003_UNIT_01_STATION_04_SAFETY_DOOR".SAFETY_DOOR.UNLOCK AND NOT "DB2120_MPP_ITC_IPC".RESET_FAULTS AND #O_BYTE_0.SEOC_WARNING);
END_REGION

REGION Network 18: UNLOCK GLOBAL REQUEST
   RUNG wire#powerrail
      Contact( "DB7003_UNIT_01_STATION_04_SAFETY_DOOR".SAFETY_DOOR.UNLOCK_MANUAL_REQUEST )
      Contact( "DB2001_MODES_GENERAL".GENERAL.MANUAL_SELECTED )
      wire#w1
      Coil( "DB7003_UNIT_01_STATION_04_SAFETY_DOOR".SAFETY_DOOR.UNLOCK_GLOBAL_REQUEST )
   END_RUNG
   RUNG wire#powerrail
      Contact( "DB7003_UNIT_01_STATION_04_SAFETY_DOOR".SAFETY_DOOR.UNLOCK_AUTO_REQUEST )
      Contact( "DB2001_MODES_GENERAL".GENERAL.AUTO_SINGLE_SEMI_SELECTED )
   END_RUNG wire#w1
   // the same network as SCL:
   "DB7003_UNIT_01_STATION_04_SAFETY_DOOR".SAFETY_DOOR.UNLOCK_GLOBAL_REQUEST := ("DB7003_UNIT_01_STATION_04_SAFETY_DOOR".SAFETY_DOOR.UNLOCK_MANUAL_REQUEST AND "DB2001_MODES_GENERAL".GENERAL.MANUAL_SELECTED) OR ("DB7003_UNIT_01_STATION_04_SAFETY_DOOR".SAFETY_DOOR.UNLOCK_AUTO_REQUEST AND "DB2001_MODES_GENERAL".GENERAL.AUTO_SINGLE_SEMI_SELECTED);
END_REGION

REGION Network 19: UNLOCK COMMAND
   RUNG wire#powerrail
      Contact( "DB7003_UNIT_01_STATION_04_SAFETY_DOOR".SAFETY_DOOR.UNLOCK_GLOBAL_REQUEST )
      wire#w1
      Contact( "DB7003_UNIT_01_STATION_04_SAFETY_DOOR".SAFETY_DOOR.PARTIAL_UNLOCK_GENERAL_CONDITIONS )
      I_Contact( "DB7003_UNIT_01_STATION_04_SAFETY_DOOR".SAFETY_DOOR.UNLOCK )
      I_Contact( "DB2120_MPP_ITC_IPC".RESET_FAULTS )
      Coil( "DB7003_UNIT_01_STATION_04_SAFETY_DOOR".SAFETY_DOOR.UNLOCK_COMMAND )
   END_RUNG
   RUNG wire#powerrail
      Contact( "DB7003_UNIT_01_STATION_04_SAFETY_DOOR".SAFETY_DOOR.UNLOCK_COMMAND )
   END_RUNG wire#w1
   // the same network as SCL:
   "DB7003_UNIT_01_STATION_04_SAFETY_DOOR".SAFETY_DOOR.UNLOCK_COMMAND := ("DB7003_UNIT_01_STATION_04_SAFETY_DOOR".SAFETY_DOOR.UNLOCK_GLOBAL_REQUEST OR "DB7003_UNIT_01_STATION_04_SAFETY_DOOR".SAFETY_DOOR.UNLOCK_COMMAND) AND "DB7003_UNIT_01_STATION_04_SAFETY_DOOR".SAFETY_DOOR.PARTIAL_UNLOCK_GENERAL_CONDITIONS AND NOT "DB7003_UNIT_01_STATION_04_SAFETY_DOOR".SAFETY_DOOR.UNLOCK AND NOT "DB2120_MPP_ITC_IPC".RESET_FAULTS;
END_REGION

REGION Network 20: UNLOCK
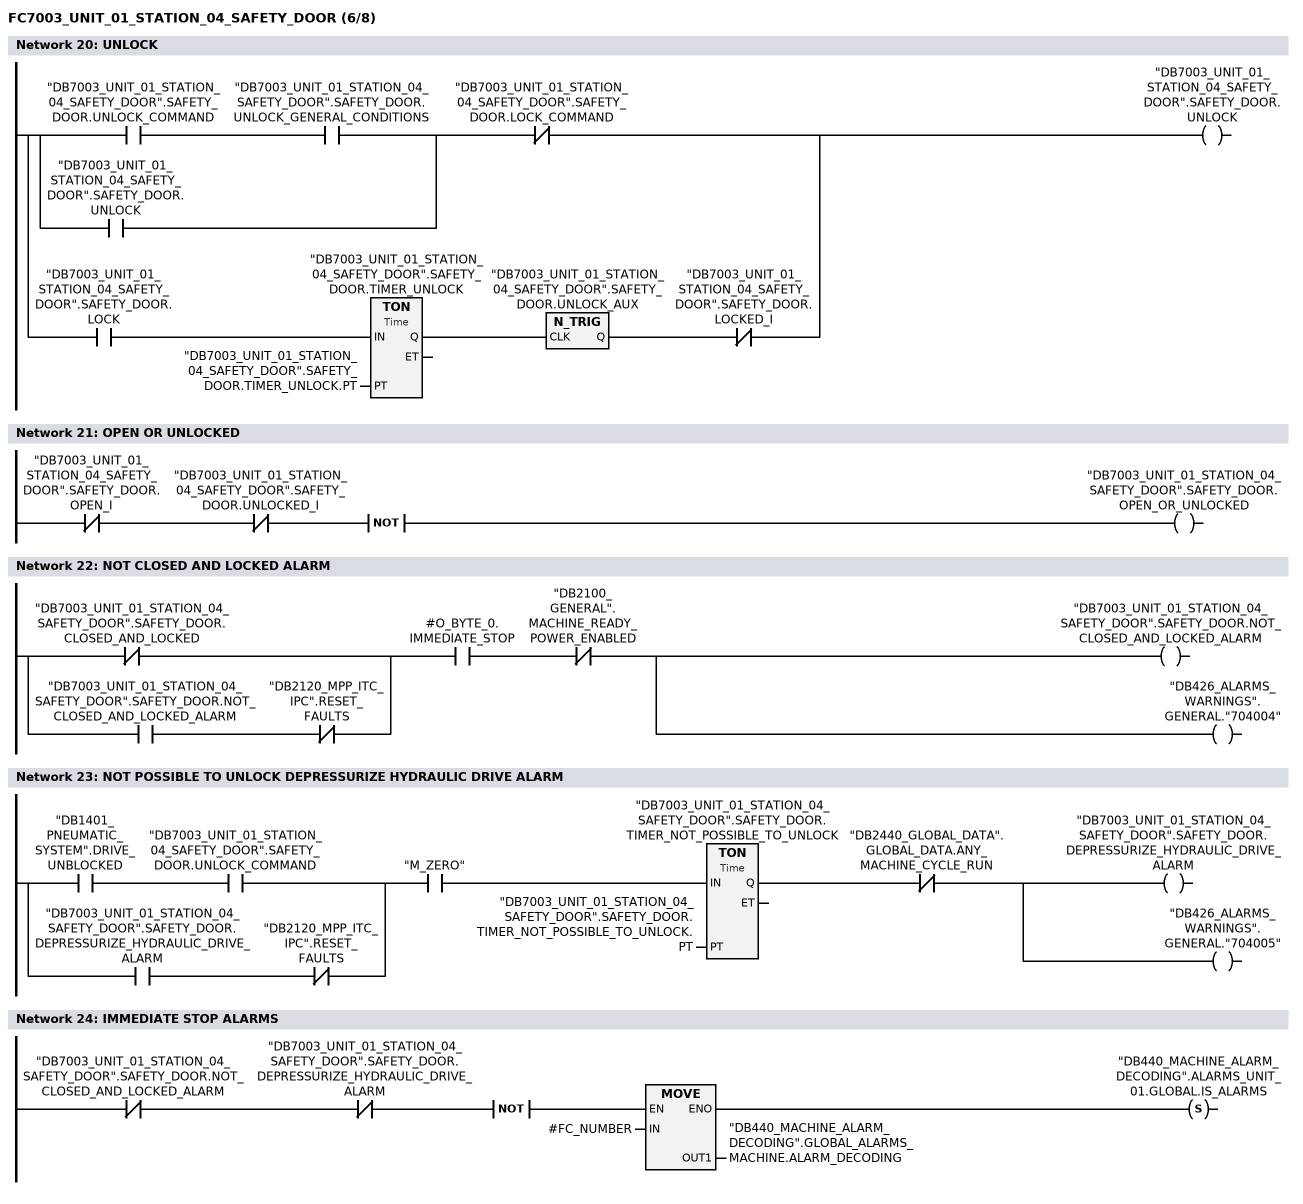
   RUNG wire#powerrail
      Contact( "DB7003_UNIT_01_STATION_04_SAFETY_DOOR".SAFETY_DOOR.UNLOCK_COMMAND )
      Contact( "DB7003_UNIT_01_STATION_04_SAFETY_DOOR".SAFETY_DOOR.UNLOCK_GENERAL_CONDITIONS )
      wire#w1
      I_Contact( "DB7003_UNIT_01_STATION_04_SAFETY_DOOR".SAFETY_DOOR.LOCK_COMMAND )
      wire#w2
      Coil( "DB7003_UNIT_01_STATION_04_SAFETY_DOOR".SAFETY_DOOR.UNLOCK )
   END_RUNG
   RUNG wire#powerrail
      Contact( "DB7003_UNIT_01_STATION_04_SAFETY_DOOR".SAFETY_DOOR.UNLOCK )
   END_RUNG wire#w1
   RUNG wire#powerrail
      Contact( "DB7003_UNIT_01_STATION_04_SAFETY_DOOR".SAFETY_DOOR.LOCK )
      { S7_Templates := "time_type := Time" } "DB7003_UNIT_01_STATION_04_SAFETY_DOOR".SAFETY_DOOR.TIMER_UNLOCK.TON(pt := "DB7003_UNIT_01_STATION_04_SAFETY_DOOR".SAFETY_DOOR.TIMER_UNLOCK.PT, et =>)
      N_Trig( "DB7003_UNIT_01_STATION_04_SAFETY_DOOR".SAFETY_DOOR.UNLOCK_AUX )
      I_Contact( "DB7003_UNIT_01_STATION_04_SAFETY_DOOR".SAFETY_DOOR.LOCKED_I )
   END_RUNG wire#w2
   // the same network as SCL:
   "DB7003_UNIT_01_STATION_04_SAFETY_DOOR".SAFETY_DOOR.TIMER_UNLOCK.TON(IN := "DB7003_UNIT_01_STATION_04_SAFETY_DOOR".SAFETY_DOOR.LOCK,
                           PT := "DB7003_UNIT_01_STATION_04_SAFETY_DOOR".SAFETY_DOOR.TIMER_UNLOCK.PT);
   #_w1 := NOT "DB7003_UNIT_01_STATION_04_SAFETY_DOOR".SAFETY_DOOR.TIMER_UNLOCK.Q AND "DB7003_UNIT_01_STATION_04_SAFETY_DOOR".SAFETY_DOOR.UNLOCK_AUX;   // falling edge
   "DB7003_UNIT_01_STATION_04_SAFETY_DOOR".SAFETY_DOOR.UNLOCK_AUX := "DB7003_UNIT_01_STATION_04_SAFETY_DOOR".SAFETY_DOOR.TIMER_UNLOCK.Q;
   "DB7003_UNIT_01_STATION_04_SAFETY_DOOR".SAFETY_DOOR.UNLOCK := ((("DB7003_UNIT_01_STATION_04_SAFETY_DOOR".SAFETY_DOOR.UNLOCK_COMMAND AND "DB7003_UNIT_01_STATION_04_SAFETY_DOOR".SAFETY_DOOR.UNLOCK_GENERAL_CONDITIONS) OR "DB7003_UNIT_01_STATION_04_SAFETY_DOOR".SAFETY_DOOR.UNLOCK) AND NOT "DB7003_UNIT_01_STATION_04_SAFETY_DOOR".SAFETY_DOOR.LOCK_COMMAND) OR (#_w1 AND NOT "DB7003_UNIT_01_STATION_04_SAFETY_DOOR".SAFETY_DOOR.LOCKED_I);
END_REGION

REGION Network 21: OPEN OR UNLOCKED
   RUNG wire#powerrail
      I_Contact( "DB7003_UNIT_01_STATION_04_SAFETY_DOOR".SAFETY_DOOR.OPEN_I )
      I_Contact( "DB7003_UNIT_01_STATION_04_SAFETY_DOOR".SAFETY_DOOR.UNLOCKED_I )
      Not()
      Coil( "DB7003_UNIT_01_STATION_04_SAFETY_DOOR".SAFETY_DOOR.OPEN_OR_UNLOCKED )
   END_RUNG
   // the same network as SCL:
   "DB7003_UNIT_01_STATION_04_SAFETY_DOOR".SAFETY_DOOR.OPEN_OR_UNLOCKED := NOT (NOT "DB7003_UNIT_01_STATION_04_SAFETY_DOOR".SAFETY_DOOR.OPEN_I AND NOT "DB7003_UNIT_01_STATION_04_SAFETY_DOOR".SAFETY_DOOR.UNLOCKED_I);
END_REGION

REGION Network 22: NOT CLOSED AND LOCKED ALARM
   RUNG wire#powerrail
      I_Contact( "DB7003_UNIT_01_STATION_04_SAFETY_DOOR".SAFETY_DOOR.CLOSED_AND_LOCKED )
      wire#w1
      Contact( #O_BYTE_0.IMMEDIATE_STOP )
      I_Contact( "DB2100_GENERAL".MACHINE_READY_POWER_ENABLED )
      wire#w2
      Coil( "DB7003_UNIT_01_STATION_04_SAFETY_DOOR".SAFETY_DOOR.NOT_CLOSED_AND_LOCKED_ALARM )
   END_RUNG
   RUNG wire#powerrail
      Contact( "DB7003_UNIT_01_STATION_04_SAFETY_DOOR".SAFETY_DOOR.NOT_CLOSED_AND_LOCKED_ALARM )
      I_Contact( "DB2120_MPP_ITC_IPC".RESET_FAULTS )
   END_RUNG wire#w1
   RUNG wire#w2
      Coil( "DB426_ALARMS_WARNINGS".GENERAL."704004" )
   END_RUNG
   // the same network as SCL:
   "DB7003_UNIT_01_STATION_04_SAFETY_DOOR".SAFETY_DOOR.NOT_CLOSED_AND_LOCKED_ALARM := (NOT "DB7003_UNIT_01_STATION_04_SAFETY_DOOR".SAFETY_DOOR.CLOSED_AND_LOCKED OR ("DB7003_UNIT_01_STATION_04_SAFETY_DOOR".SAFETY_DOOR.NOT_CLOSED_AND_LOCKED_ALARM AND NOT "DB2120_MPP_ITC_IPC".RESET_FAULTS)) AND #O_BYTE_0.IMMEDIATE_STOP AND NOT "DB2100_GENERAL".MACHINE_READY_POWER_ENABLED;
   "DB426_ALARMS_WARNINGS".GENERAL."704004" := "DB7003_UNIT_01_STATION_04_SAFETY_DOOR".SAFETY_DOOR.NOT_CLOSED_AND_LOCKED_ALARM;
END_REGION

REGION Network 23: NOT POSSIBLE TO UNLOCK DEPRESSURIZE HYDRAULIC DRIVE ALARM
   RUNG wire#powerrail
      Contact( "DB1401_PNEUMATIC_SYSTEM".DRIVE_UNBLOCKED )
      Contact( "DB7003_UNIT_01_STATION_04_SAFETY_DOOR".SAFETY_DOOR.UNLOCK_COMMAND )
      wire#w1
      Contact( "M_ZERO" )
      { S7_Templates := "time_type := Time" } "DB7003_UNIT_01_STATION_04_SAFETY_DOOR".SAFETY_DOOR.TIMER_NOT_POSSIBLE_TO_UNLOCK.TON(pt := "DB7003_UNIT_01_STATION_04_SAFETY_DOOR".SAFETY_DOOR.TIMER_NOT_POSSIBLE_TO_UNLOCK.PT, et =>)
      I_Contact( "DB2440_GLOBAL_DATA".GLOBAL_DATA.ANY_MACHINE_CYCLE_RUN )
      wire#w2
      Coil( "DB7003_UNIT_01_STATION_04_SAFETY_DOOR".SAFETY_DOOR.DEPRESSURIZE_HYDRAULIC_DRIVE_ALARM )
   END_RUNG
   RUNG wire#powerrail
      Contact( "DB7003_UNIT_01_STATION_04_SAFETY_DOOR".SAFETY_DOOR.DEPRESSURIZE_HYDRAULIC_DRIVE_ALARM )
      I_Contact( "DB2120_MPP_ITC_IPC".RESET_FAULTS )
   END_RUNG wire#w1
   RUNG wire#w2
      Coil( "DB426_ALARMS_WARNINGS".GENERAL."704005" )
   END_RUNG
   // the same network as SCL:
   "DB7003_UNIT_01_STATION_04_SAFETY_DOOR".SAFETY_DOOR.TIMER_NOT_POSSIBLE_TO_UNLOCK.TON(IN := (("DB1401_PNEUMATIC_SYSTEM".DRIVE_UNBLOCKED AND "DB7003_UNIT_01_STATION_04_SAFETY_DOOR".SAFETY_DOOR.UNLOCK_COMMAND) OR ("DB7003_UNIT_01_STATION_04_SAFETY_DOOR".SAFETY_DOOR.DEPRESSURIZE_HYDRAULIC_DRIVE_ALARM AND NOT "DB2120_MPP_ITC_IPC".RESET_FAULTS)) AND "M_ZERO",
                           PT := "DB7003_UNIT_01_STATION_04_SAFETY_DOOR".SAFETY_DOOR.TIMER_NOT_POSSIBLE_TO_UNLOCK.PT);
   "DB7003_UNIT_01_STATION_04_SAFETY_DOOR".SAFETY_DOOR.DEPRESSURIZE_HYDRAULIC_DRIVE_ALARM := "DB7003_UNIT_01_STATION_04_SAFETY_DOOR".SAFETY_DOOR.TIMER_NOT_POSSIBLE_TO_UNLOCK.Q AND NOT "DB2440_GLOBAL_DATA".GLOBAL_DATA.ANY_MACHINE_CYCLE_RUN;
   "DB426_ALARMS_WARNINGS".GENERAL."704005" := "DB7003_UNIT_01_STATION_04_SAFETY_DOOR".SAFETY_DOOR.DEPRESSURIZE_HYDRAULIC_DRIVE_ALARM;
END_REGION

REGION Network 24: IMMEDIATE STOP ALARMS
   RUNG wire#powerrail
      I_Contact( "DB7003_UNIT_01_STATION_04_SAFETY_DOOR".SAFETY_DOOR.NOT_CLOSED_AND_LOCKED_ALARM )
      I_Contact( "DB7003_UNIT_01_STATION_04_SAFETY_DOOR".SAFETY_DOOR.DEPRESSURIZE_HYDRAULIC_DRIVE_ALARM )
      Not()
      { S7_GenerateENO := "TRUE" } Move(in := #FC_NUMBER, out1 => "DB440_MACHINE_ALARM_DECODING".GLOBAL_ALARMS_MACHINE.ALARM_DECODING)
      S_Coil( "DB440_MACHINE_ALARM_DECODING".ALARMS_UNIT_01.GLOBAL.IS_ALARMS )
   END_RUNG
   // the same network as SCL:
   // ENO of a box is taken as its EN; it also drops when the box reports an error
   IF NOT (NOT "DB7003_UNIT_01_STATION_04_SAFETY_DOOR".SAFETY_DOOR.NOT_CLOSED_AND_LOCKED_ALARM AND NOT "DB7003_UNIT_01_STATION_04_SAFETY_DOOR".SAFETY_DOOR.DEPRESSURIZE_HYDRAULIC_DRIVE_ALARM) THEN
       "DB440_MACHINE_ALARM_DECODING".GLOBAL_ALARMS_MACHINE.ALARM_DECODING := #FC_NUMBER;
       "DB440_MACHINE_ALARM_DECODING".ALARMS_UNIT_01.GLOBAL.IS_ALARMS := TRUE;
   END_IF;
END_REGION

REGION Network 25: UNLOCK REQUEST WARNING
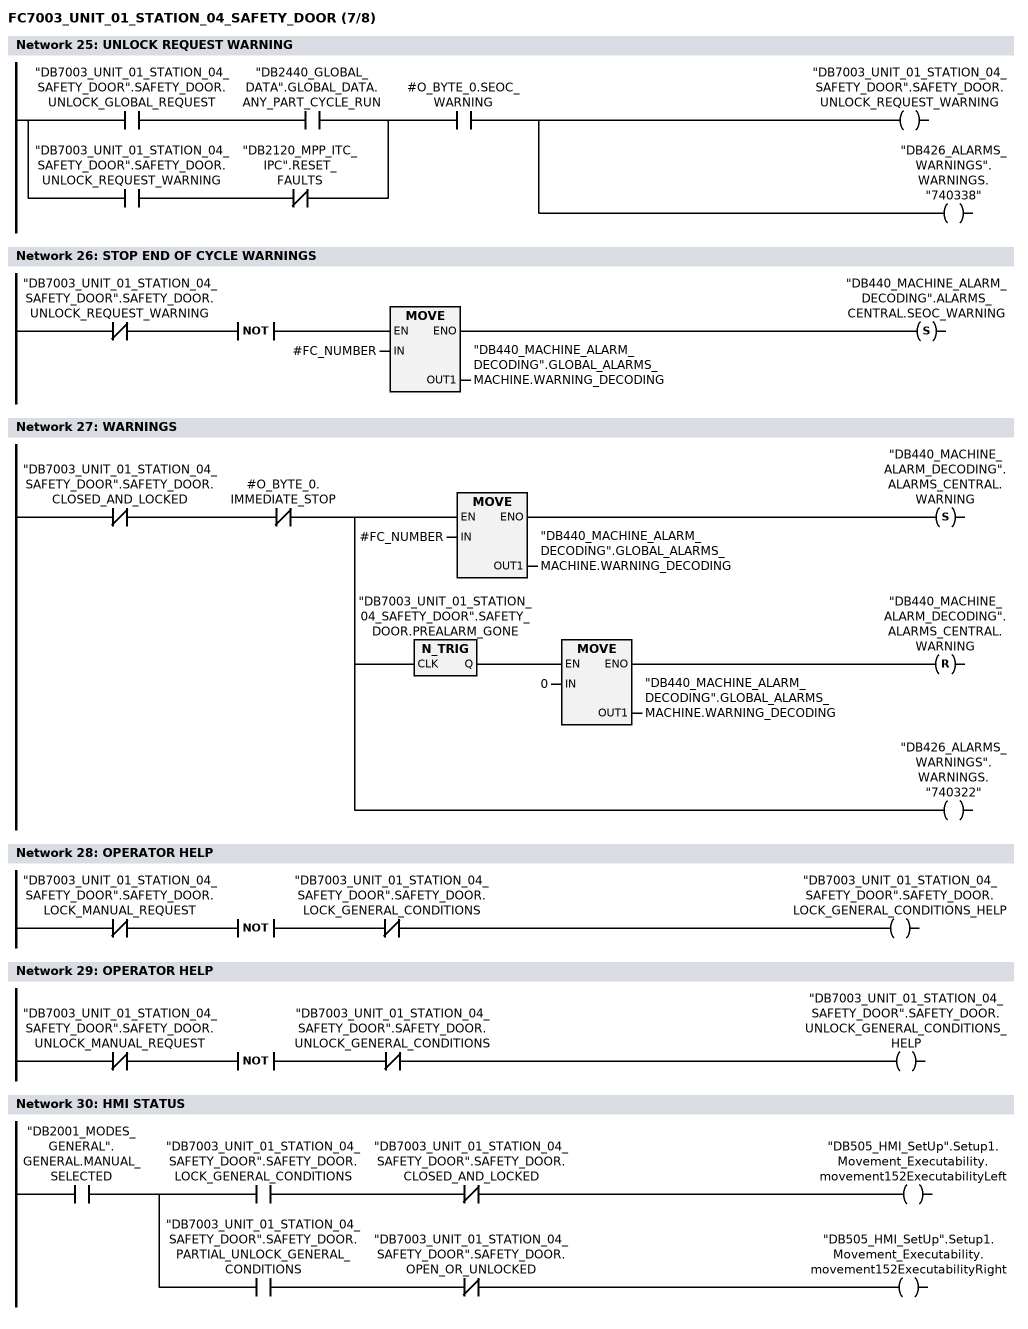
   RUNG wire#powerrail
      Contact( "DB7003_UNIT_01_STATION_04_SAFETY_DOOR".SAFETY_DOOR.UNLOCK_GLOBAL_REQUEST )
      Contact( "DB2440_GLOBAL_DATA".GLOBAL_DATA.ANY_PART_CYCLE_RUN )
      wire#w1
      Contact( #O_BYTE_0.SEOC_WARNING )
      wire#w2
      Coil( "DB7003_UNIT_01_STATION_04_SAFETY_DOOR".SAFETY_DOOR.UNLOCK_REQUEST_WARNING )
   END_RUNG
   RUNG wire#powerrail
      Contact( "DB7003_UNIT_01_STATION_04_SAFETY_DOOR".SAFETY_DOOR.UNLOCK_REQUEST_WARNING )
      I_Contact( "DB2120_MPP_ITC_IPC".RESET_FAULTS )
   END_RUNG wire#w1
   RUNG wire#w2
      Coil( "DB426_ALARMS_WARNINGS".WARNINGS."740338" )
   END_RUNG
   // the same network as SCL:
   "DB7003_UNIT_01_STATION_04_SAFETY_DOOR".SAFETY_DOOR.UNLOCK_REQUEST_WARNING := (("DB7003_UNIT_01_STATION_04_SAFETY_DOOR".SAFETY_DOOR.UNLOCK_GLOBAL_REQUEST AND "DB2440_GLOBAL_DATA".GLOBAL_DATA.ANY_PART_CYCLE_RUN) OR ("DB7003_UNIT_01_STATION_04_SAFETY_DOOR".SAFETY_DOOR.UNLOCK_REQUEST_WARNING AND NOT "DB2120_MPP_ITC_IPC".RESET_FAULTS)) AND #O_BYTE_0.SEOC_WARNING;
   "DB426_ALARMS_WARNINGS".WARNINGS."740338" := "DB7003_UNIT_01_STATION_04_SAFETY_DOOR".SAFETY_DOOR.UNLOCK_REQUEST_WARNING;
END_REGION

REGION Network 26: STOP END OF CYCLE WARNINGS
   RUNG wire#powerrail
      I_Contact( "DB7003_UNIT_01_STATION_04_SAFETY_DOOR".SAFETY_DOOR.UNLOCK_REQUEST_WARNING )
      Not()
      { S7_GenerateENO := "TRUE" } Move(in := #FC_NUMBER, out1 => "DB440_MACHINE_ALARM_DECODING".GLOBAL_ALARMS_MACHINE.WARNING_DECODING)
      S_Coil( "DB440_MACHINE_ALARM_DECODING".ALARMS_CENTRAL.SEOC_WARNING )
   END_RUNG
   // the same network as SCL:
   // ENO of a box is taken as its EN; it also drops when the box reports an error
   IF NOT (NOT "DB7003_UNIT_01_STATION_04_SAFETY_DOOR".SAFETY_DOOR.UNLOCK_REQUEST_WARNING) THEN
       "DB440_MACHINE_ALARM_DECODING".GLOBAL_ALARMS_MACHINE.WARNING_DECODING := #FC_NUMBER;
       "DB440_MACHINE_ALARM_DECODING".ALARMS_CENTRAL.SEOC_WARNING := TRUE;
   END_IF;
END_REGION

REGION Network 27: WARNINGS
   RUNG wire#powerrail
      I_Contact( "DB7003_UNIT_01_STATION_04_SAFETY_DOOR".SAFETY_DOOR.CLOSED_AND_LOCKED )
      I_Contact( #O_BYTE_0.IMMEDIATE_STOP )
      wire#w1
      { S7_GenerateENO := "TRUE" } Move(in := #FC_NUMBER, out1 => "DB440_MACHINE_ALARM_DECODING".GLOBAL_ALARMS_MACHINE.WARNING_DECODING)
      S_Coil( "DB440_MACHINE_ALARM_DECODING".ALARMS_CENTRAL.WARNING )
   END_RUNG
   RUNG wire#w1
      N_Trig( "DB7003_UNIT_01_STATION_04_SAFETY_DOOR".SAFETY_DOOR.PREALARM_GONE )
      { S7_GenerateENO := "TRUE" } Move(in := 0, out1 => "DB440_MACHINE_ALARM_DECODING".GLOBAL_ALARMS_MACHINE.WARNING_DECODING)
      R_Coil( "DB440_MACHINE_ALARM_DECODING".ALARMS_CENTRAL.WARNING )
   END_RUNG
   RUNG wire#w1
      Coil( "DB426_ALARMS_WARNINGS".WARNINGS."740322" )
   END_RUNG
   // the same network as SCL:
   // ENO of a box is taken as its EN; it also drops when the box reports an error
   #_w1 := NOT "DB7003_UNIT_01_STATION_04_SAFETY_DOOR".SAFETY_DOOR.CLOSED_AND_LOCKED AND NOT #O_BYTE_0.IMMEDIATE_STOP;
   IF #_w1 THEN
       "DB440_MACHINE_ALARM_DECODING".GLOBAL_ALARMS_MACHINE.WARNING_DECODING := #FC_NUMBER;
       "DB440_MACHINE_ALARM_DECODING".ALARMS_CENTRAL.WARNING := TRUE;
   END_IF;
   #_w2 := NOT #_w1 AND "DB7003_UNIT_01_STATION_04_SAFETY_DOOR".SAFETY_DOOR.PREALARM_GONE;   // falling edge
   "DB7003_UNIT_01_STATION_04_SAFETY_DOOR".SAFETY_DOOR.PREALARM_GONE := #_w1;
   IF #_w2 THEN
       "DB440_MACHINE_ALARM_DECODING".GLOBAL_ALARMS_MACHINE.WARNING_DECODING := 0;
       "DB440_MACHINE_ALARM_DECODING".ALARMS_CENTRAL.WARNING := FALSE;
   END_IF;
   "DB426_ALARMS_WARNINGS".WARNINGS."740322" := #_w1;
END_REGION

REGION Network 28: OPERATOR HELP
   RUNG wire#powerrail
      I_Contact( "DB7003_UNIT_01_STATION_04_SAFETY_DOOR".SAFETY_DOOR.LOCK_MANUAL_REQUEST )
      Not()
      I_Contact( "DB7003_UNIT_01_STATION_04_SAFETY_DOOR".SAFETY_DOOR.LOCK_GENERAL_CONDITIONS )
      Coil( "DB7003_UNIT_01_STATION_04_SAFETY_DOOR".SAFETY_DOOR.LOCK_GENERAL_CONDITIONS_HELP )
   END_RUNG
   // the same network as SCL:
   "DB7003_UNIT_01_STATION_04_SAFETY_DOOR".SAFETY_DOOR.LOCK_GENERAL_CONDITIONS_HELP := NOT (NOT "DB7003_UNIT_01_STATION_04_SAFETY_DOOR".SAFETY_DOOR.LOCK_MANUAL_REQUEST) AND NOT "DB7003_UNIT_01_STATION_04_SAFETY_DOOR".SAFETY_DOOR.LOCK_GENERAL_CONDITIONS;
END_REGION

REGION Network 29: OPERATOR HELP
   RUNG wire#powerrail
      I_Contact( "DB7003_UNIT_01_STATION_04_SAFETY_DOOR".SAFETY_DOOR.UNLOCK_MANUAL_REQUEST )
      Not()
      I_Contact( "DB7003_UNIT_01_STATION_04_SAFETY_DOOR".SAFETY_DOOR.UNLOCK_GENERAL_CONDITIONS )
      Coil( "DB7003_UNIT_01_STATION_04_SAFETY_DOOR".SAFETY_DOOR.UNLOCK_GENERAL_CONDITIONS_HELP )
   END_RUNG
   // the same network as SCL:
   "DB7003_UNIT_01_STATION_04_SAFETY_DOOR".SAFETY_DOOR.UNLOCK_GENERAL_CONDITIONS_HELP := NOT (NOT "DB7003_UNIT_01_STATION_04_SAFETY_DOOR".SAFETY_DOOR.UNLOCK_MANUAL_REQUEST) AND NOT "DB7003_UNIT_01_STATION_04_SAFETY_DOOR".SAFETY_DOOR.UNLOCK_GENERAL_CONDITIONS;
END_REGION

REGION Network 30: HMI STATUS
   RUNG wire#powerrail
      Contact( "DB2001_MODES_GENERAL".GENERAL.MANUAL_SELECTED )
      wire#w1
      Contact( "DB7003_UNIT_01_STATION_04_SAFETY_DOOR".SAFETY_DOOR.LOCK_GENERAL_CONDITIONS )
      I_Contact( "DB7003_UNIT_01_STATION_04_SAFETY_DOOR".SAFETY_DOOR.CLOSED_AND_LOCKED )
      Coil( "DB505_HMI_SetUp".Setup1.Movement_Executability.movement152ExecutabilityLeft )
   END_RUNG
   RUNG wire#w1
      Contact( "DB7003_UNIT_01_STATION_04_SAFETY_DOOR".SAFETY_DOOR.PARTIAL_UNLOCK_GENERAL_CONDITIONS )
      I_Contact( "DB7003_UNIT_01_STATION_04_SAFETY_DOOR".SAFETY_DOOR.OPEN_OR_UNLOCKED )
      Coil( "DB505_HMI_SetUp".Setup1.Movement_Executability.movement152ExecutabilityRight )
   END_RUNG
   // the same network as SCL:
   "DB505_HMI_SetUp".Setup1.Movement_Executability.movement152ExecutabilityLeft := "DB2001_MODES_GENERAL".GENERAL.MANUAL_SELECTED AND "DB7003_UNIT_01_STATION_04_SAFETY_DOOR".SAFETY_DOOR.LOCK_GENERAL_CONDITIONS AND NOT "DB7003_UNIT_01_STATION_04_SAFETY_DOOR".SAFETY_DOOR.CLOSED_AND_LOCKED;
   "DB505_HMI_SetUp".Setup1.Movement_Executability.movement152ExecutabilityRight := "DB2001_MODES_GENERAL".GENERAL.MANUAL_SELECTED AND "DB7003_UNIT_01_STATION_04_SAFETY_DOOR".SAFETY_DOOR.PARTIAL_UNLOCK_GENERAL_CONDITIONS AND NOT "DB7003_UNIT_01_STATION_04_SAFETY_DOOR".SAFETY_DOOR.OPEN_OR_UNLOCKED;
END_REGION

REGION Network 31: HMI STATUS
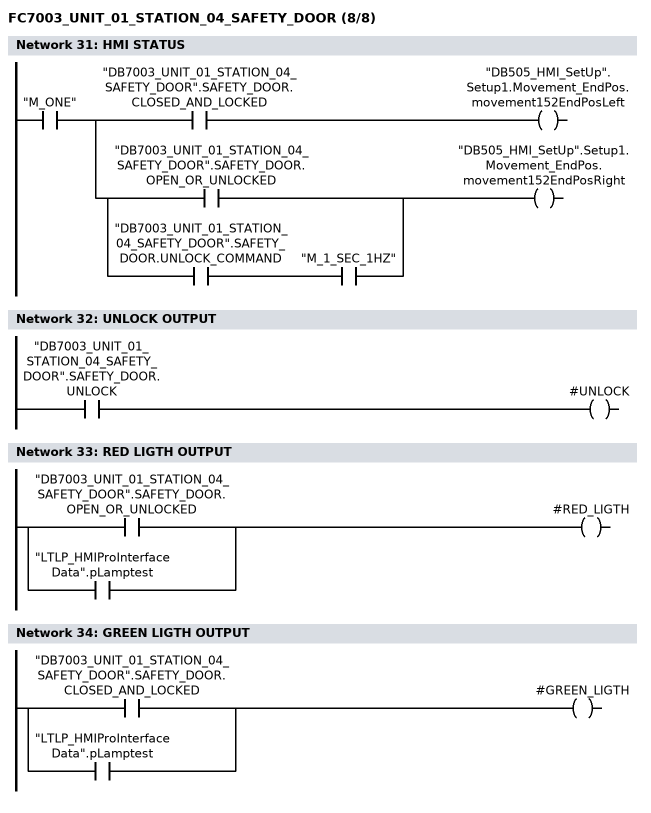
   RUNG wire#powerrail
      Contact( "M_ONE" )
      wire#w1
      Contact( "DB7003_UNIT_01_STATION_04_SAFETY_DOOR".SAFETY_DOOR.CLOSED_AND_LOCKED )
      Coil( "DB505_HMI_SetUp".Setup1.Movement_EndPos.movement152EndPosLeft )
   END_RUNG
   RUNG wire#w1
      Contact( "DB7003_UNIT_01_STATION_04_SAFETY_DOOR".SAFETY_DOOR.OPEN_OR_UNLOCKED )
      wire#w2
      Coil( "DB505_HMI_SetUp".Setup1.Movement_EndPos.movement152EndPosRight )
   END_RUNG
   RUNG wire#w1
      Contact( "DB7003_UNIT_01_STATION_04_SAFETY_DOOR".SAFETY_DOOR.UNLOCK_COMMAND )
      Contact( "M_1_SEC_1HZ" )
   END_RUNG wire#w2
   // the same network as SCL:
   "DB505_HMI_SetUp".Setup1.Movement_EndPos.movement152EndPosLeft := "M_ONE" AND "DB7003_UNIT_01_STATION_04_SAFETY_DOOR".SAFETY_DOOR.CLOSED_AND_LOCKED;
   "DB505_HMI_SetUp".Setup1.Movement_EndPos.movement152EndPosRight := "M_ONE" AND ("DB7003_UNIT_01_STATION_04_SAFETY_DOOR".SAFETY_DOOR.OPEN_OR_UNLOCKED OR ("DB7003_UNIT_01_STATION_04_SAFETY_DOOR".SAFETY_DOOR.UNLOCK_COMMAND AND "M_1_SEC_1HZ"));
END_REGION

REGION Network 32: UNLOCK OUTPUT
   RUNG wire#powerrail
      Contact( "DB7003_UNIT_01_STATION_04_SAFETY_DOOR".SAFETY_DOOR.UNLOCK )
      Coil( #UNLOCK )
   END_RUNG
   // the same network as SCL:
   #UNLOCK := "DB7003_UNIT_01_STATION_04_SAFETY_DOOR".SAFETY_DOOR.UNLOCK;
END_REGION

REGION Network 33: RED LIGTH OUTPUT
   RUNG wire#powerrail
      Contact( "DB7003_UNIT_01_STATION_04_SAFETY_DOOR".SAFETY_DOOR.OPEN_OR_UNLOCKED )
      wire#w1
      Coil( #RED_LIGTH )
   END_RUNG
   RUNG wire#powerrail
      Contact( "LTLP_HMIProInterfaceData".pLamptest )
   END_RUNG wire#w1
   // the same network as SCL:
   #RED_LIGTH := "DB7003_UNIT_01_STATION_04_SAFETY_DOOR".SAFETY_DOOR.OPEN_OR_UNLOCKED OR "LTLP_HMIProInterfaceData".pLamptest;
END_REGION

REGION Network 34: GREEN LIGTH OUTPUT
   RUNG wire#powerrail
      Contact( "DB7003_UNIT_01_STATION_04_SAFETY_DOOR".SAFETY_DOOR.CLOSED_AND_LOCKED )
      wire#w1
      Coil( #GREEN_LIGTH )
   END_RUNG
   RUNG wire#powerrail
      Contact( "LTLP_HMIProInterfaceData".pLamptest )
   END_RUNG wire#w1
   // the same network as SCL:
   #GREEN_LIGTH := "DB7003_UNIT_01_STATION_04_SAFETY_DOOR".SAFETY_DOOR.CLOSED_AND_LOCKED OR "LTLP_HMIProInterfaceData".pLamptest;
END_REGION
END_FUNCTION
